# EPICS autosave request: ipApp/Db/Thorlabs_SC10_settings.req
$(P)$(S):UpdateRBVs.SCAN
$(P)$(S):ShutTime
$(P)$(S):OpenTime
$(P)$(S):Reps
$(P)$(S):Mode
$(P)$(S):ExtTriggerOutMode
$(P)$(S):TriggerMode
$(P)$(S):Enable
